// TIA Portal project "THU_LIMES_RoboticMillingSystem_20241015_V18" (V18)

(* hardware
DEVICE "S7-1200 station_1"  S7-1200 Station
   slot 0: "Rack_0"  S7-1200 Rack  Rack  V1.0
   slot 1: "PLC_1"  CPU 1214C DC/DC/DC  6ES7 214-1AG40-0XB0  V4.5
   slot 2: "DI 8x24VDC/DQ 8xRelay_1"  SM 1223 DI8/DQ8 x relay  6ES7 223-1PH32-0XB0  V2.0
   slot 3: "AQ 2x14BIT_1"  SM 1232 AQ2  6ES7 232-4HB32-0XB0  V2.1
DEVICE "GSD device_1"  GSD.Device.PN
   slot 0: "机架"  Rack  V1.0
   slot 0: "RobotBasicIO"  BASIC V1.4  888-3  V1.4
      slot 0: "Robot Basic Device"  Robot Basic Device  888-3  V1.4
      slot 1: "PROFINET Interface"  PROFINET Interface
         slot 1: "Network Port"  Network Port
   slot 1: "DI 64 bytes_1"  DI 64 bytes
      slot 0: "DI 64 bytes"  DI 64 bytes
   slot 2: "DO 64 bytes_1"  DO 64 bytes
      slot 0: "DO 64 bytes"  DO 64 bytes
*)

// ===== PLC "PLC_1"  CPU 1214C DC/DC/DC =====
// protected blocks, not shown: "电主轴速度调节", "电主轴速度采集"

VAR_GLOBAL   // PLC tag table "默认变量表"
   "A相" AT %I0.0 : Bool;
   "B相" AT %I0.1 : Bool;
   "换刀信号" AT %I0.2 : Bool;
   "拉刀气压监控" AT %I0.3 : Bool;
   "卸刀气压监控" AT %I0.4 : Bool;
   "拉刀信号反馈" AT %I0.5 : Bool;
   "卸刀信号反馈" AT %I0.6 : Bool;
   "A_7" AT %I0.7 : Bool;
   "启动按钮" AT %I1.0 : Bool;
   "复位按钮" AT %I1.1 : Bool;
   "A_10" AT %I1.2 : Bool;
   "A_11" AT %I1.3 : Bool;
   "A_12" AT %I1.4 : Bool;
   "A_13" AT %I1.5 : Bool;
   "变频器停止信号" AT %I2.0 : Bool;
   "变频器启动信号" AT %I2.1 : Bool;
   "A_16" AT %I2.2 : Bool;
   "A_17" AT %I2.3 : Bool;
   "HSC_1_INC_采集值" AT %ID1000 : DInt;
   "实时速度输出" AT %QW112 : Int;
   "启动指示灯" AT %Q0.0 : Bool;
   "复位指示灯" AT %Q0.1 : Bool;
   "运行指示灯" AT %Q0.2 : Bool;
   "故障指示灯" AT %Q0.4 : Bool;
   "拉卸刀电磁阀" AT %Q0.5 : Bool;
   "气源总开关" AT %Q0.6 : Bool;
   "吹尘电磁阀" AT %Q0.7 : Bool;
   "换刀按钮灯" AT %Q1.0 : Bool;
   "B_9" AT %Q1.1 : Bool;
   "System_Byte" AT %MB1 : Byte;
   "FirstScan" AT %M1.0 : Bool;
   "DiagStatusUpdate" AT %M1.1 : Bool;
   "AlwaysTRUE" AT %M1.2 : Bool;
   "AlwaysFALSE" AT %M1.3 : Bool;
   "Clock_Byte" AT %MB0 : Byte;
   "Clock_10Hz" AT %M0.0 : Bool;
   "Clock_5Hz" AT %M0.1 : Bool;
   "Clock_2.5Hz" AT %M0.2 : Bool;
   "Clock_2Hz" AT %M0.3 : Bool;
   "Clock_1.25Hz" AT %M0.4 : Bool;
   "Clock_1Hz" AT %M0.5 : Bool;
   "Clock_0.625Hz" AT %M0.6 : Bool;
   "Clock_0.5Hz" AT %M0.7 : Bool;
   "电主轴启动" AT %M100.0 : Bool;
   "电主轴停止" AT %M100.1 : Bool;
   "变频器停" AT %M100.2 : Bool;
   "变频器停沿信号" AT %M100.3 : Bool;
   "C#_停沿信号" AT %M100.4 : Bool;
   "电主轴运行指示灯" AT %M100.5 : Bool;
   "HSC_Done" AT %M200.0 : Bool;
   "HSC_Busy" AT %M200.1 : Bool;
   "HSC_Error" AT %M200.2 : Bool;
   "HSC_Status" AT %MW300 : Word;
   "C_4" AT %M200.4 : Bool;
   "C_5" AT %M200.5 : Bool;
   "C_6" AT %M200.6 : Bool;
   "C_7" AT %M200.7 : Bool;
   "GetInteruptData" AT %MD300 : DInt;
   "Frenqucy" AT %MD304 : DInt;
   "Rpm_Second" AT %MD308 : DInt;
   "Rpm_Minute" AT %MD312 : DInt;
   "C_12" AT %MD316 : DInt;
   "C_13" AT %MD320 : DInt;
   "INC_COUNTER" AT %MD1000 : DWord;
   "FromABB" AT %ID100 : DWord;
   "ActualVaule" AT %MD500 : DWord;
   "Tag_1" AT %MW500 : Word;
   "ABB_TO_PLC" AT %I105.0 : Bool;
   "ABB设置主轴转速权限信号上升沿" AT %M1100.0 : Bool;
   "ABB换刀信号" AT %I104.1 : Bool;
   "C#_Working" AT %M1100.1 : Bool;
   "变频器启动" AT %Q10.0 : Bool;
   "变频器停止" AT %Q10.1 : Bool;
   "Robot_变频器启动" AT %I104.2 : Bool;
   "Robot_变频器停止" AT %I104.3 : Bool;
   "变频运行" AT %Q2.6 : Bool;
   "Robot_变频停止" AT %Q2.7 : Bool;
   "Speed_Second" AT %MD108 : Real;
   "Tag_6" AT %M1000.0 : Bool;
   "Tag_8" AT %MD5000 : DInt;
   "Tag_9" AT %MD104 : Real;
   "HSC_perSecond" AT %MD112 : Real;
   "Speed_perMin" AT %MD120 : Real;
   "ABB_send_speed" AT %MD130 : Real;
   "ABB设置主轴转速权限转换信号" AT %M1100.2 : Bool;
   "C#_WorkDone" AT %M1100.3 : Bool;
   "ABB设置主轴转速权限信号下降沿" AT %M1100.4 : Bool;
   "Tag_6(1)" AT %M1100.5 : Bool;
   "C#_send_speed" AT %MD134 : Real;
   "ABB设置主轴转速权限信号" AT %I104.0 : Bool;
   "断开Robot控制" AT %M1100.6 : Bool;
   "上位机锁定换刀按钮" AT %M1000.7 : Bool;
   "拉刀指示灯" AT %Q0.3 : Bool;
   "ABB_Speed" AT %MD260 : Real;
   "ABB_Speed_temp" AT %MD264 : Real;
END_VAR

TYPE "电机运行及调速控制"
VERSION : 0.1
   STRUCT
      设定运行时间 : Time;
      给定频率 : Real;
   END_STRUCT;
END_TYPE

DATA_BLOCK "Send_HMI_Data"   // DB1
{ S7_Optimized_Access := 'FALSE' }
VERSION : 0.1
   VAR
      Static_1 : Bool;
      Static_2 : Bool;
      电主轴实时转速反馈 : DInt;
      HMI_频率输入 : Real;
      HMI_给定频率 : Real;
   END_VAR
BEGIN
END_DATA_BLOCK

DATA_BLOCK "电主轴运行数据"   // DB2
{ S7_Optimized_Access := 'TRUE' }
VERSION : 0.1
   VAR
      电主轴 : "电机运行及调速控制";
      FromABB : Real;
      FromABBDATA : Array[0..3] of Byte;
      Temp_1 : DWord;
      Temp_2 : DWord;
      Temp_3 : Real;
   END_VAR
BEGIN
END_DATA_BLOCK

DATA_BLOCK "DB_HSC"   // DB3
{ S7_Optimized_Access := 'TRUE' }
VERSION : 0.1
   VAR
      Count : HSC_Count;
      HSC_脉冲转换值 : Real;
      HSC_Speed_perScond : Real;
      HSC_Raio_result_DINT : DInt;
      TempSpeed_Real : Real;
      TempSpeed_INT : Int;
      SendSpeed_INT : Int;
   END_VAR
BEGIN
   // Count.CurrentCount : 高速计数器的当前值
   // Count.EnHSC : 启用高速计数器
   // Count.EnSync : 同步输入(I0.7与EnSync同时为1，同步输入才生效)
END_DATA_BLOCK

DATA_BLOCK "C#_Data"   // DB11
{ S7_Optimized_Access := 'FALSE' }
VERSION : 0.1
   VAR
      Send_RotateSpeed : String[8];   // 编码器转速转发到上位机
      RcvData : String[8];
      TSEND_DONE : Bool;
      TSEND_BUSY : Bool;
      TSEND_ERROR : Bool;
      TSEND_STATUS : Word;
      TRCV_C_DONE : Bool;
      TRCV_C_BUSY : Bool;
      TRCV_C_ERROR : Bool;
      TRCV_C_STATUS : Word;
      TRCV_C_RCV_LEN : UInt;
      NDR : Bool;
      S_CONV_Spindle_Motion : String;   // 来自上位机的主轴启停信号
      "S_CONV_#" : String := '#';   // 上位机结束符
      "0S_CONV_Spindle_RotateSpeed" : String;   // 编码器转速转换值
      GetLenSpeed : Int := 5;
      GetPosSpeed : Int := 1;
      GetstringSpeed : String;   // 读取上位机的转速
      GetstringMotion : String;   // 读取上位机的启停信号
      GetLenBool : Int := 1;
      GetPosBool : Int := 7;
      S_CONV_Int_Speed : Int;   // 分割出的转速值
      S_CONV_Int_Motion : Int;   // 分割触出的启停信号
      Right_Num : Int := 2;   // 读取字符串右侧的数据，右往左2个字符
      Temp1 : Real;
      Temp3 : DInt;
      Temp4 : Real;
      Temp2 : Real;
      Fake_Spindle_Speed_Polyfit : Int;
      Send_Speed_Spindle_Real : Int;
      Send_Speed_Spindle_Int : Int;
   END_VAR
BEGIN
END_DATA_BLOCK

// folder: System blocks/Program resources

DATA_BLOCK "PLC_1_Receive_DB"   // DB10
{ S7_Optimized_Access := 'TRUE' }
AUTHOR : SIMATIC
FAMILY : MC7Plus
NAME : TC_IP_v4
VERSION : 1.0
// stored: InstanceOfName TCON_IP_v4
"TCON_IP_v4"
BEGIN
   ID := 1;
   InterfaceId := 64;
   LocalPort := 2000;
END_DATA_BLOCK

// folder: (top level)

FUNCTION "气动控制" : Void   // FC1, SCL
{ S7_Optimized_Access := 'TRUE' }
VERSION : 0.1
   VAR_INPUT
      "biTO/TI_Monitor" : Bool;   // 左侧真空压力表
      biCL_Monitor : Bool;   // 右侧压力表
      biTI_SigFeedBack : Bool;   // 拉刀信号反馈
      biTO_SigFeedBack : Bool;   // 卸刀信号反馈
      biExchangeSignal : Bool;   // 换刀信号
      HMI_biExchangeSignal : Bool;
      Robot_Tool_Change : Bool;   // 机器人请求换刀
      Button_Tool_Change : Bool;   // 按钮换刀
      Tool_Change_Complete : Bool;   // 换刀完成信号
   END_VAR
   VAR_OUTPUT
      "boTO/TI" : Bool;   // 拉刀卸刀
      boAirControl : Bool;   // 气源控制
      boCL : Bool;   // 吹尘
      "boTO/TI_Light" : Bool;   // 换刀按钮灯
      "boRed&buzzer" : Bool;
   END_VAR
   VAR_TEMP
      T1_OK : Bool;   // 拉刀成功
   END_VAR
BEGIN

   #boAirControl := "AlwaysTRUE"; //开机气源一直为TRUE状态，气封接头一直通气
   //IF #Robot_Tool_Change OR #Button_Tool_Change THEN
   //#boCL := 0; //换刀时，断开总气源
   //ELSE
   // "IEC_Timer_0_DB".TON(IN:=#Tool_Change_Complete,
   //  PT:=T#1s,
   //  Q=>#boCL);
   //END_IF;

   //换刀逻辑

   IF NOT  "变频运行" THEN

   IF #biExchangeSignal OR #HMI_biExchangeSignal THEN  //换刀信号为TRUE
       #"boTO/TI" := TRUE;   //换刀电磁阀置1
       //#"boRed&buzzer" := "Clock_0.5Hz";
       IF #biTI_SigFeedBack AND NOT #biTO_SigFeedBack THEN//拉刀为TRUE，卸刀为FALSE，换刀成功
           #T1_OK := TRUE; //换刀成功，
       ELSE
           #T1_OK := FALSE;
           #"boRed&buzzer" := "Clock_1Hz";
       END_IF;
   END_IF;

   END_IF;


   //中心吹尘
   IF NOT #biTI_SigFeedBack AND #biTO_SigFeedBack THEN
       #boCL := TRUE;
   END_IF;

   IF #biTI_SigFeedBack AND NOT #biTO_SigFeedBack THEN
       #boCL := FALSE;
   END_IF;
END_FUNCTION

FUNCTION "报警" : Void   // FC2, SCL
{ S7_Optimized_Access := 'TRUE' }
VERSION : 0.1
   VAR_INPUT
      biTI_Alarm : Bool;
      biTO_Alarm : Bool;
      biReset : Bool;
      biConverter_start : Bool;
   END_VAR
   VAR_OUTPUT
      boRedAlarm : Bool;
   END_VAR
BEGIN
   //压力表报警
   IF #biConverter_start THEN
       IF NOT #biTI_Alarm OR NOT #biTO_Alarm THEN
           #boRedAlarm := TRUE;
       END_IF;
   END_IF;

   IF #biReset THEN
       #boRedAlarm := FALSE;
   END_IF;
END_FUNCTION

FUNCTION "SpindleMotion" : Void   // FC3, SCL
{ S7_Optimized_Access := 'TRUE' }
VERSION : 0.1
BEGIN
END_FUNCTION

ORGANIZATION_BLOCK "Main"   // OB1, LAD, ProgramCycle
TITLE = "Main Program Sweep (Cycle)"
{ S7_Optimized_Access := 'TRUE' }
VERSION : 0.1
   VAR_INPUT
      Initial_Call : Bool;   // Initial call of this OB
      Remanence : Bool;   // =True, if remanent data are available
   END_VAR
   VAR_TEMP   // added for the SCL form of the ladder/FBD networks
      _w1 : Bool;
      _w2 : Bool;
      _w3 : Bool;
      _w4 : Bool;
   END_VAR
BEGIN

REGION Network 1: 指示灯
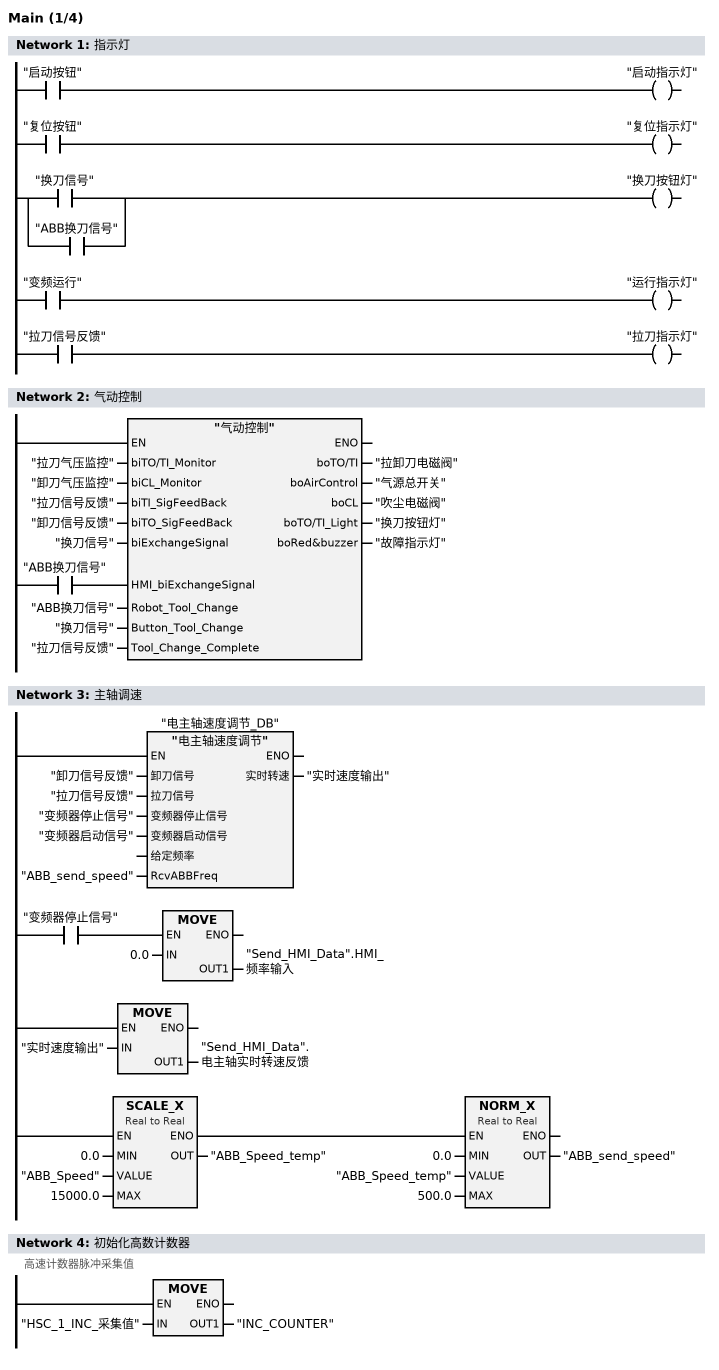
   RUNG wire#powerrail
      Contact( "启动按钮" )
      Coil( "启动指示灯" )
   END_RUNG
   RUNG wire#powerrail
      Contact( "复位按钮" )
      Coil( "复位指示灯" )
   END_RUNG
   RUNG wire#powerrail
      Contact( "换刀信号" )
      wire#w1
      Coil( "换刀按钮灯" )
   END_RUNG
   RUNG wire#powerrail
      Contact( "ABB换刀信号" )
   END_RUNG wire#w1
   RUNG wire#powerrail
      Contact( "变频运行" )
      Coil( "运行指示灯" )
   END_RUNG
   RUNG wire#powerrail
      Contact( "拉刀信号反馈" )
      Coil( "拉刀指示灯" )
   END_RUNG
   // the same network as SCL:
   "启动指示灯" := "启动按钮";
   "复位指示灯" := "复位按钮";
   "换刀按钮灯" := "换刀信号" OR "ABB换刀信号";
   "运行指示灯" := "变频运行";
   "拉刀指示灯" := "拉刀信号反馈";
END_REGION

REGION Network 2: 气动控制
   RUNG wire#powerrail
      "气动控制"(HMI_biExchangeSignal := wire#w1, "biTO/TI_Monitor" := "拉刀气压监控", biCL_Monitor := "卸刀气压监控", biTI_SigFeedBack := "拉刀信号反馈", biTO_SigFeedBack := "卸刀信号反馈", biExchangeSignal := "换刀信号", Robot_Tool_Change := "ABB换刀信号", Button_Tool_Change := "换刀信号", Tool_Change_Complete := "拉刀信号反馈", "boTO/TI" => "拉卸刀电磁阀", boAirControl => "气源总开关", boCL => "吹尘电磁阀", "boTO/TI_Light" => "换刀按钮灯", "boRed&buzzer" => "故障指示灯")
   END_RUNG
   RUNG wire#powerrail
      Contact( "ABB换刀信号" )
   END_RUNG wire#w1
   // the same network as SCL:
   "气动控制"("biTO/TI_Monitor" := "拉刀气压监控",
          biCL_Monitor := "卸刀气压监控",
          biTI_SigFeedBack := "拉刀信号反馈",
          biTO_SigFeedBack := "卸刀信号反馈",
          biExchangeSignal := "换刀信号",
          HMI_biExchangeSignal := "ABB换刀信号",
          Robot_Tool_Change := "ABB换刀信号",
          Button_Tool_Change := "换刀信号",
          Tool_Change_Complete := "拉刀信号反馈",
          "boTO/TI" => "拉卸刀电磁阀",
          boAirControl => "气源总开关",
          boCL => "吹尘电磁阀",
          "boTO/TI_Light" => "换刀按钮灯",
          "boRed&buzzer" => "故障指示灯");
END_REGION

REGION Network 3: 主轴调速
   RUNG wire#powerrail
      "电主轴速度调节_DB"(卸刀信号 := "卸刀信号反馈", 拉刀信号 := "拉刀信号反馈", 变频器停止信号 := "变频器停止信号", 变频器启动信号 := "变频器启动信号", 给定频率 :=, RcvABBFreq := "ABB_send_speed", 实时转速 => "实时速度输出")
   END_RUNG
   RUNG wire#powerrail
      Contact( "变频器停止信号" )
      Move(in := 0.0, out1 => "Send_HMI_Data".HMI_频率输入)
   END_RUNG
   RUNG wire#powerrail
      Move(in := "实时速度输出", out1 => "Send_HMI_Data".电主轴实时转速反馈)
   END_RUNG
   RUNG wire#powerrail
      { S7_Templates := "[SrcType := Real, DestType := Real]" } Scale(min := 0.0, value := "ABB_Speed", max := 15000.0, out => "ABB_Speed_temp")
      { S7_Templates := "[SrcType := Real, DestType := Real]" } Normalize(min := 0.0, value := "ABB_Speed_temp", max := 500.0, out => "ABB_send_speed")
   END_RUNG
   // the same network as SCL:
   "电主轴速度调节_DB"(卸刀信号 := "卸刀信号反馈",   // "电主轴速度调节"
                拉刀信号 := "拉刀信号反馈",
                变频器停止信号 := "变频器停止信号",
                变频器启动信号 := "变频器启动信号",
                RcvABBFreq := "ABB_send_speed",
                实时转速 => "实时速度输出");
   IF "变频器停止信号" THEN "Send_HMI_Data".HMI_频率输入 := 0.0; END_IF;
   "Send_HMI_Data".电主轴实时转速反馈 := "实时速度输出";
   "ABB_Speed_temp" := SCALE_X(MIN := 0.0, VALUE := "ABB_Speed", MAX := 15000.0);
   "ABB_send_speed" := NORM_X(MIN := 0.0, VALUE := "ABB_Speed_temp", MAX := 500.0);
END_REGION

REGION Network 4: 初始化高数计数器
   // 高速计数器脉冲采集值
   RUNG wire#powerrail
      Move(in := "HSC_1_INC_采集值", out1 => "INC_COUNTER")
   END_RUNG
   // the same network as SCL:
   "INC_COUNTER" := "HSC_1_INC_采集值";
END_REGION

REGION Network 5: 故障报警
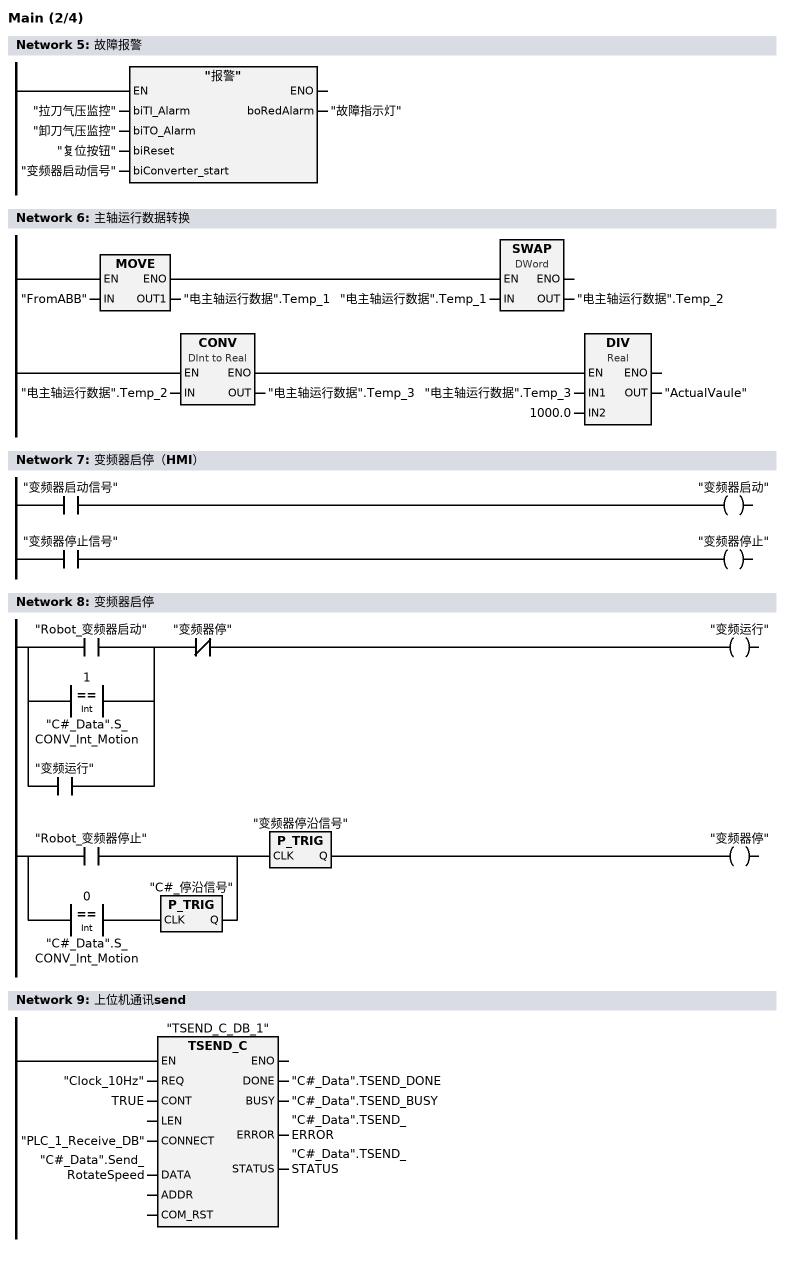
   RUNG wire#powerrail
      "报警"(biTI_Alarm := "拉刀气压监控", biTO_Alarm := "卸刀气压监控", biReset := "复位按钮", biConverter_start := "变频器启动信号", boRedAlarm => "故障指示灯")
   END_RUNG
   // the same network as SCL:
   "报警"(biTI_Alarm := "拉刀气压监控",
        biTO_Alarm := "卸刀气压监控",
        biReset := "复位按钮",
        biConverter_start := "变频器启动信号",
        boRedAlarm => "故障指示灯");
END_REGION

REGION Network 6: 主轴运行数据转换
   "电主轴运行数据".Temp_1 := "FromABB";
   "电主轴运行数据".Temp_2 := SWAP("电主轴运行数据".Temp_1);
   "电主轴运行数据".Temp_3 := DINT_TO_REAL("电主轴运行数据".Temp_2);
   "ActualVaule" := "电主轴运行数据".Temp_3 / 1000.0;
END_REGION

REGION Network 7: 变频器启停（HMI）
   RUNG wire#powerrail
      Contact( "变频器启动信号" )
      Coil( "变频器启动" )
   END_RUNG
   RUNG wire#powerrail
      Contact( "变频器停止信号" )
      Coil( "变频器停止" )
   END_RUNG
   // the same network as SCL:
   "变频器启动" := "变频器启动信号";
   "变频器停止" := "变频器停止信号";
END_REGION

REGION Network 8: 变频器启停
   RUNG wire#powerrail
      Contact( "Robot_变频器启动" )
      wire#w1
      I_Contact( "变频器停" )
      Coil( "变频运行" )
   END_RUNG
   RUNG wire#powerrail
      { S7_Templates := "SrcType := Int" } EQ_Contact(in1 := 1, in2 := "C#_Data".S_CONV_Int_Motion)
   END_RUNG wire#w1
   RUNG wire#powerrail
      Contact( "变频运行" )
   END_RUNG wire#w1
   RUNG wire#powerrail
      Contact( "Robot_变频器停止" )
      wire#w2
      P_Trig( "变频器停沿信号" )
      Coil( "变频器停" )
   END_RUNG
   RUNG wire#powerrail
      { S7_Templates := "SrcType := Int" } EQ_Contact(in1 := 0, in2 := "C#_Data".S_CONV_Int_Motion)
      P_Trig( "C#_停沿信号" )
   END_RUNG wire#w2
   // the same network as SCL:
   "变频运行" := ("Robot_变频器启动" OR (1 = "C#_Data".S_CONV_Int_Motion) OR "变频运行") AND NOT "变频器停";
   #_w1 := 0 = "C#_Data".S_CONV_Int_Motion;
   #_w2 := #_w1 AND NOT "C#_停沿信号";   // rising edge
   "C#_停沿信号" := #_w1;
   #_w3 := "Robot_变频器停止" OR #_w2;
   #_w4 := #_w3 AND NOT "变频器停沿信号";   // rising edge
   "变频器停沿信号" := #_w3;
   "变频器停" := #_w4;
END_REGION

REGION Network 9: 上位机通讯send
   "TSEND_C_DB_1"(REQ := "Clock_10Hz",   // TSEND_C
                  CONT := TRUE,
                  CONNECT := "PLC_1_Receive_DB",
                  DATA := "C#_Data".Send_RotateSpeed,
                  DONE => "C#_Data".TSEND_DONE,
                  BUSY => "C#_Data".TSEND_BUSY,
                  ERROR => "C#_Data".TSEND_ERROR,
                  STATUS => "C#_Data".TSEND_STATUS);
END_REGION

REGION Network 10: 上位机通讯Trcv
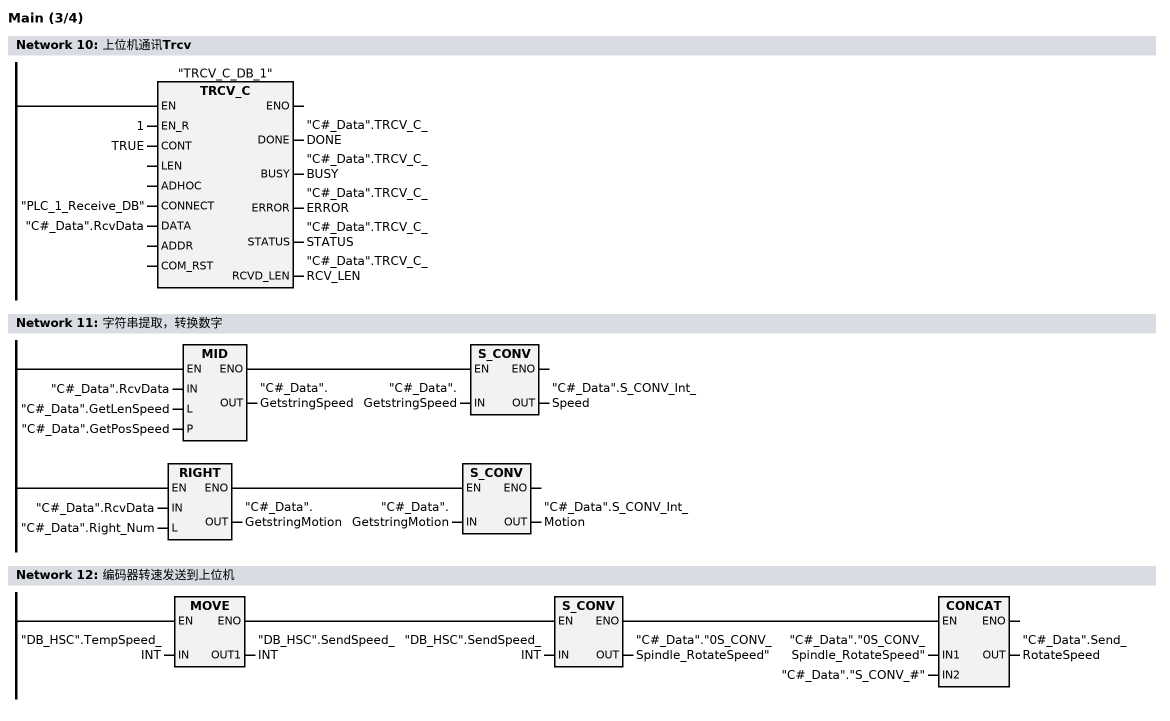
   "TRCV_C_DB_1"(EN_R := 1,   // TRCV_C
                 CONT := TRUE,
                 CONNECT := "PLC_1_Receive_DB",
                 DATA := "C#_Data".RcvData,
                 DONE => "C#_Data".TRCV_C_DONE,
                 BUSY => "C#_Data".TRCV_C_BUSY,
                 ERROR => "C#_Data".TRCV_C_ERROR,
                 STATUS => "C#_Data".TRCV_C_STATUS,
                 RCVD_LEN => "C#_Data".TRCV_C_RCV_LEN);
END_REGION

REGION Network 11: 字符串提取，转换数字
   "C#_Data".GetstringSpeed := MID(IN := "C#_Data".RcvData,
                           L := "C#_Data".GetLenSpeed,
                           P := "C#_Data".GetPosSpeed);
   "C#_Data".S_CONV_Int_Speed := S_CONV(IN := "C#_Data".GetstringSpeed);
   "C#_Data".GetstringMotion := RIGHT(IN := "C#_Data".RcvData, L := "C#_Data".Right_Num);
   "C#_Data".S_CONV_Int_Motion := S_CONV(IN := "C#_Data".GetstringMotion);
END_REGION

REGION Network 12: 编码器转速发送到上位机
   "DB_HSC".SendSpeed_INT := "DB_HSC".TempSpeed_INT;
   "C#_Data"."0S_CONV_Spindle_RotateSpeed" := S_CONV(IN := "DB_HSC".SendSpeed_INT);
   "C#_Data".Send_RotateSpeed := CONCAT(IN1 := "C#_Data"."0S_CONV_Spindle_RotateSpeed",
                           IN2 := "C#_Data"."S_CONV_#");
END_REGION

REGION Network 13: Robot/上位机互锁
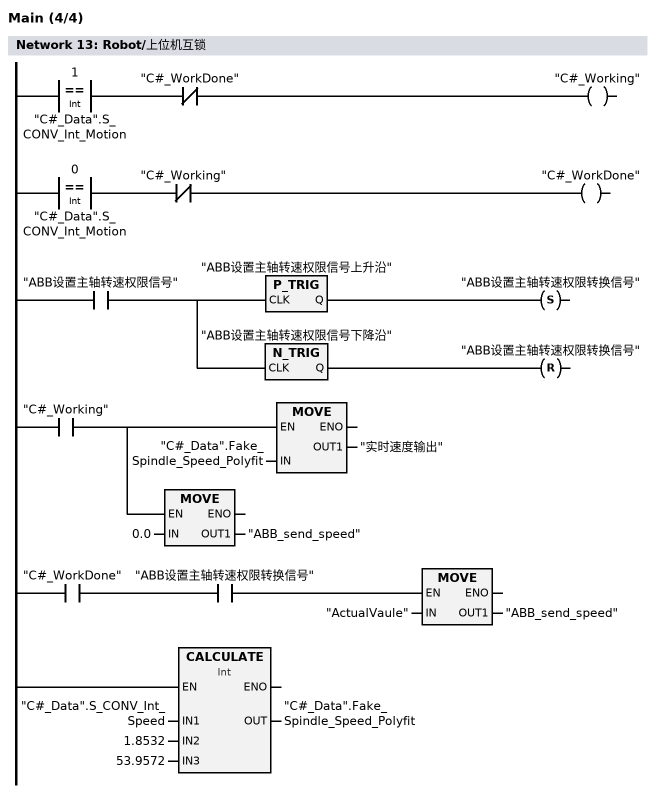
   RUNG wire#powerrail
      { S7_Templates := "SrcType := Int" } EQ_Contact(in1 := 1, in2 := "C#_Data".S_CONV_Int_Motion)
      I_Contact( "C#_WorkDone" )
      Coil( "C#_Working" )
   END_RUNG
   RUNG wire#powerrail
      { S7_Templates := "SrcType := Int" } EQ_Contact(in1 := 0, in2 := "C#_Data".S_CONV_Int_Motion)
      I_Contact( "C#_Working" )
      Coil( "C#_WorkDone" )
   END_RUNG
   RUNG wire#powerrail
      Contact( "ABB设置主轴转速权限信号" )
      wire#w1
      P_Trig( "ABB设置主轴转速权限信号上升沿" )
      S_Coil( "ABB设置主轴转速权限转换信号" )
   END_RUNG
   RUNG wire#w1
      N_Trig( "ABB设置主轴转速权限信号下降沿" )
      R_Coil( "ABB设置主轴转速权限转换信号" )
   END_RUNG
   RUNG wire#powerrail
      Contact( "C#_Working" )
      wire#w2
      Move(in := "C#_Data".Fake_Spindle_Speed_Polyfit, out1 => "实时速度输出")
   END_RUNG
   RUNG wire#w2
      Move(in := 0.0, out1 => "ABB_send_speed")
   END_RUNG
   RUNG wire#powerrail
      Contact( "C#_WorkDone" )
      Contact( "ABB设置主轴转速权限转换信号" )
      Move(in := "ActualVaule", out1 => "ABB_send_speed")
   END_RUNG
   RUNG wire#powerrail
      { S7_Templates := "SrcType := Int"; S7_Expression := "IN1*IN2+IN3" } Calculate(in1 := "C#_Data".S_CONV_Int_Speed, in2 := 1.8532, in3 := 53.9572, out => "C#_Data".Fake_Spindle_Speed_Polyfit)
   END_RUNG
   // the same network as SCL:
   "C#_Working" := (1 = "C#_Data".S_CONV_Int_Motion) AND NOT "C#_WorkDone";
   "C#_WorkDone" := (0 = "C#_Data".S_CONV_Int_Motion) AND NOT "C#_Working";
   #_w1 := "ABB设置主轴转速权限信号" AND NOT "ABB设置主轴转速权限信号上升沿";   // rising edge
   "ABB设置主轴转速权限信号上升沿" := "ABB设置主轴转速权限信号";
   IF #_w1 THEN "ABB设置主轴转速权限转换信号" := TRUE; END_IF;
   #_w2 := NOT "ABB设置主轴转速权限信号" AND "ABB设置主轴转速权限信号下降沿";   // falling edge
   "ABB设置主轴转速权限信号下降沿" := "ABB设置主轴转速权限信号";
   IF #_w2 THEN "ABB设置主轴转速权限转换信号" := FALSE; END_IF;
   IF "C#_Working" THEN
       "实时速度输出" := "C#_Data".Fake_Spindle_Speed_Polyfit;
       "ABB_send_speed" := 0.0;
   END_IF;
   IF "C#_WorkDone" AND "ABB设置主轴转速权限转换信号" THEN "ABB_send_speed" := "ActualVaule"; END_IF;
   "C#_Data".Fake_Spindle_Speed_Polyfit := "C#_Data".S_CONV_Int_Speed*1.8532+53.9572;
END_REGION
END_ORGANIZATION_BLOCK

ORGANIZATION_BLOCK "Cyclic interrupt"   // OB30, LAD, CyclicInterrupt
{ S7_Optimized_Access := 'TRUE' }
VERSION : 0.1
   VAR_INPUT
      Initial_Call : Bool;   // Initial call of this OB
      Event_Count : Int;   // Events discarded
   END_VAR
BEGIN

REGION Network 1: 高数计数器初始化
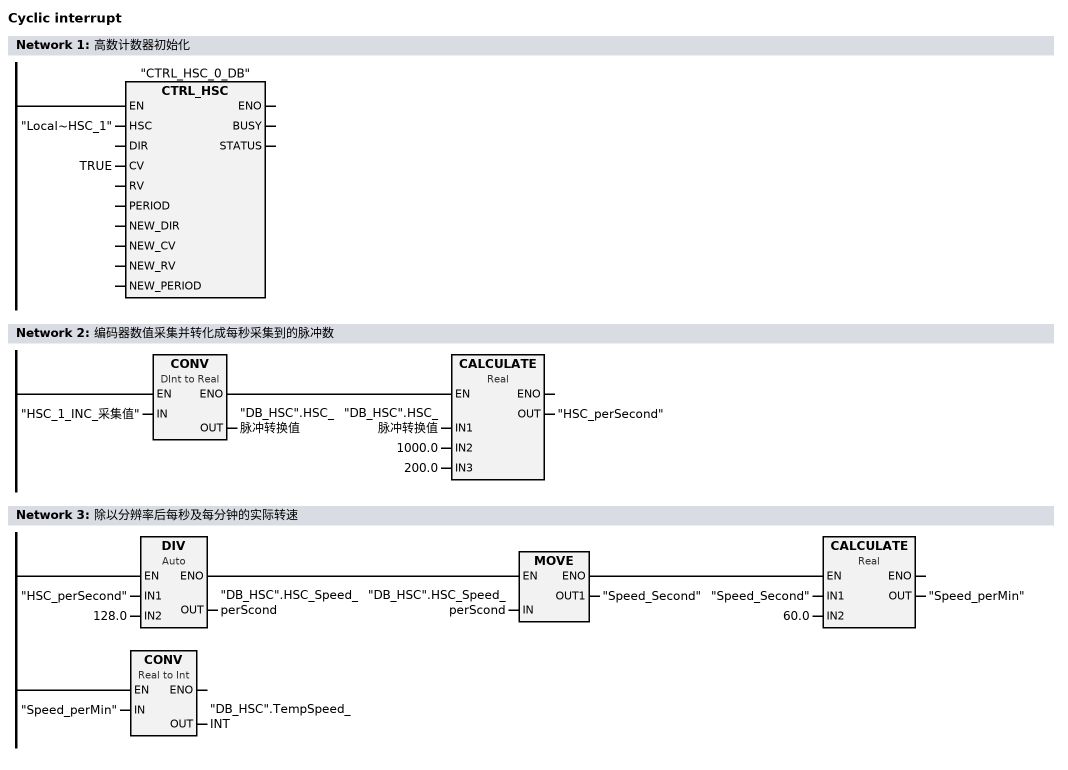
   "CTRL_HSC_0_DB"(HSC := "Local~HSC_1", CV := TRUE);   // CTRL_HSC
END_REGION

REGION Network 2: 编码器数值采集并转化成每秒采集到的脉冲数
   RUNG wire#powerrail
      { S7_Templates := "[SrcType := DInt, DestType := Real]" } Convert(in := "HSC_1_INC_采集值", out => "DB_HSC".HSC_脉冲转换值)
      { S7_Templates := "SrcType := Real"; S7_Expression := "(IN1*IN2)/IN3" } Calculate(in1 := "DB_HSC".HSC_脉冲转换值, in2 := 1000.0, in3 := 200.0, out => "HSC_perSecond")
   END_RUNG
   // the same network as SCL:
   "DB_HSC".HSC_脉冲转换值 := DINT_TO_REAL("HSC_1_INC_采集值");
   "HSC_perSecond" := ("DB_HSC".HSC_脉冲转换值*1000.0)/200.0;
END_REGION

REGION Network 3: 除以分辨率后每秒及每分钟的实际转速
   RUNG wire#powerrail
      Div(in1 := "HSC_perSecond", in2 := 128.0, out => "DB_HSC".HSC_Speed_perScond)
      Move(in := "DB_HSC".HSC_Speed_perScond, out1 => "Speed_Second")
      { S7_Templates := "SrcType := Real"; S7_Expression := "IN1*IN2" } Calculate(in1 := "Speed_Second", in2 := 60.0, out => "Speed_perMin")
   END_RUNG
   RUNG wire#powerrail
      { S7_Templates := "[SrcType := Real, DestType := Int]" } Convert(in := "Speed_perMin", out => "DB_HSC".TempSpeed_INT)
   END_RUNG
   // the same network as SCL:
   "DB_HSC".HSC_Speed_perScond := "HSC_perSecond" / 128.0;
   "Speed_Second" := "DB_HSC".HSC_Speed_perScond;
   "Speed_perMin" := "Speed_Second"*60.0;
   "DB_HSC".TempSpeed_INT := REAL_TO_INT("Speed_perMin");
END_REGION
END_ORGANIZATION_BLOCK